Fanuc KAREL source: MIRROR.kl

PROGRAM T
%NOLOCKGROUP
VAR
 v0 : POSITION
 v1 : POSITION
 v2 : BOOLEAN
 res : XYZWPREXT
BEGIN
 res = MIRROR(v0, v1, v2)
END T
